// TIA Portal V21 export
FUNCTION "AllarmiMacchina_010102" : Void   // FC151, LAD
{ S7_Optimized_Access := 'TRUE' }
// stored: SetENOAutomatically false
   VAR_TEMP
      "Counter" : Int;
   END_VAR
   VAR CONSTANT
      K_NumAllarmeGenerico_DeltaP_Filtri : Int := 1;
      K_NumAllarmeGenerico_DeltaT_UscitaSterilizzazione : Int := 2;
      K_NumAllarmeGenerico_DeltaT_UscitaSosta : Int := 3;
   END_VAR
BEGIN

REGION Network 1 (SCL): Instasamento FILTRI (Delta Pres)
   "GestAnalogica_Delta"(K_Analogica_1 := "K_Analogica_PressioneIngressoFiltriProdotto",
                         K_Analogica_2 := "K_Analogica_PressioneUscitaFiltriProdotto",
                         K_Zona := "K_Zona_Sterilizzatore",
                         K_NumAllarmeGenerico := #K_NumAllarmeGenerico_DeltaP_Filtri,
                         MassimaDistanza := 2.0,
                         Ritardo:="TimerZona".DeltaP_Filtri);
END_REGION

REGION Network 2 (SCL): Sonde PT100 processo e storicizzazione (Delta Temp)
   "GestAnalogica_Delta"(K_Analogica_1 := "K_Analogica_TemperaturaUscitaSterilizzatoreProcesso",
                         K_Analogica_2 := "K_Analogica_TemperaturaUscitaSterilizzatoreStoricizzare",
                         K_Zona := "K_Zona_Sterilizzatore",
                         K_NumAllarmeGenerico := #K_NumAllarmeGenerico_DeltaT_UscitaSterilizzazione,
                         MassimaDistanza := 1.0,
                         Ritardo:="TimerZona"."DeltaT_UscitaSterilizzazione");

   "GestAnalogica_Delta"(K_Analogica_1 := "K_Analogica_TemperaturaUscitaSosta",
                         K_Analogica_2 := "K_Analogica_TemperaturaUscitaSostaStoricizzazione",
                         K_Zona := "K_Zona_Sterilizzatore",
                         K_NumAllarmeGenerico := #K_NumAllarmeGenerico_DeltaT_UscitaSosta,
                         MassimaDistanza := 1.0,
                         Ritardo:="TimerZona".DeltaT_UscitaSosta);
END_REGION

REGION Network 3 (SCL): Gestione generica degli allarmi
   REGION Gestione degli allarmi specifici e generali della zona
       FOR #Counter := 1 TO 15 DO
           "GestAllarme_Std"(GestioneSirena := True,
                             Allarme := "Zona".Z[K_Zona_Sterilizzatore].Allarmi.AG[#Counter],
                             NumAllarme := #Counter,
                             K_Zona := "K_Zona_Sterilizzatore",
                             WordHmi := "Zona".Z[K_Zona_Sterilizzatore].Allarmi.WordHMI_AG);
       END_FOR;
   END_REGION ;
END_REGION
END_FUNCTION
